(*	This FB is used for a single output solenoid 
	It uses the single input to say when Extended  	
	It starts assuming retracted and the output off.
*)
FUNCTION_BLOCK FB_Contactor_With_Single_Feedback EXTENDS FB_ComponentBase IMPLEMENTS I_Contactor
VAR
    //Output
    Output 				AT %Q* : BOOL;
//	FeedBackExtended	AT %I* : BOOL;	//This could be an sensor FB
	ExtendedSensor		:FB_DigitalSensor		:= (Name := 'Sensor', DebounceMode := E_DebounceMode.SimpleFlickerFilter, DebounceTime := T#250MS, Inverted    := FALSE, SimulationInput:= FALSE, SimulationMode := E_SensorSimulationMode.InputDriven) ;

    // Internal variables
    _ExtendRequest  : BOOL;
    _RetractRequest : BOOL;
    _Extended       : BOOL;
    _Retracted      : BOOL;
    _Extending      : BOOL;
    _Retracting     : BOOL;
    _ExtendTime     : LREAL := 1000; // Default time 1s
    _RetractTime    : LREAL := 1000; // Default time 1s

    // Timer for Extend/Retract
    Extend_TON    : TON;
    Retract_TON   : TON;
    Extend_RTRIG  : R_TRIG;
    Retract_RTRIG : R_TRIG;

    //HMI 
    Contactor_HMI : ST_Contactor_HMI;
END_VAR

METHOD PROTECTED CreateEvents
VAR_INPUT
END_VAR
SUPER^.CreateEvents();
END_METHOD

METHOD CyclicLogic
//One shot the requests
Extend_RTRIG(CLK := _ExtendRequest);
Retract_RTRIG(CLK := _RetractRequest);

//Handle Extend
IF Extend_RTRIG.Q THEN
    Output          := TRUE;
    _Extending      := TRUE;
    _Retracting     := FALSE;
    _Retracted      := FALSE;
    _RetractRequest := FALSE;
END_IF

//Handle Retract
IF Retract_RTRIG.Q THEN
    Output         := FALSE;
    _Extending     := FALSE;
    _Retracting    := TRUE;
    _Extended      := FALSE;
    _ExtendRequest := FALSE;
END_IF

//Handle the time to Extend/Retract
Extend_TON(IN := _Extending, PT := LREAL_TO_TIME(_ExtendTime));
Retract_TON(IN := _Retracting, PT := LREAL_TO_TIME(_RetractTime));
IF ExtendedSensor.Active THEN
    _Extended  := TRUE;
    _Extending := FALSE;
END_IF

IF Retract_TON.Q AND NOT ExtendedSensor.Active THEN
    _Retracted  := TRUE;
    _Retracting := FALSE;
END_IF

SUPER^.CyclicLogic();
END_METHOD

METHOD Extend
_ExtendRequest  := TRUE;
_RetractRequest := FALSE;
END_METHOD

PROPERTY Extended : BOOL
GET
Extended := _Extended;
END_GET
END_PROPERTY

PROPERTY ExtendTime : LREAL
GET
ExtendTime := _ExtendTime;
END_GET
SET
END_SET
END_PROPERTY

METHOD PROTECTED HMICommunication
VAR_INPUT
END_VAR
SUPER^.HMICommunication();

//Handle the requests to extend and retract
IF ComponentBase_HMI.Status.HMIControlAvailable THEN
    IF Contactor_HMI.Command.Extend THEN
        Extend();
    ELSIF Contactor_HMI.Command.Retract THEN
        Retract();
    END_IF
END_IF

//Update HMI status info
Contactor_HMI.Status.Extended    := _Extended;
Contactor_HMI.Status.Extending   := _Extending;
Contactor_HMI.Status.Retracted   := _Retracted;
Contactor_HMI.Status.Retracting  := _Retracting;
Contactor_HMI.Config.ExtendTime  := _ExtendTime;
Contactor_HMI.Config.RetractTime := _RetractTime;
END_METHOD

//! @summary Basic component initialization logic
METHOD PROTECTED Initialize : BOOL;

//! @description This method is called by <c>CyclicLogic()</c> as required
//Set the Contactor to retracted
IF Output THEN
    _Extended  := TRUE;
    _Retracted := FALSE;
ELSE
    _Extended  := FALSE;
    _Retracted := TRUE;
END_IF

_Extending      := FALSE;
_ExtendRequest  := FALSE;
_Retracting     := FALSE;
_RetractRequest := FALSE;

//Call base class Initialize
Initialize := SUPER^.Initialize();
END_METHOD

METHOD PROTECTED Monitoring
VAR_INPUT
END_VAR
_Busy    := _Extending OR _Retracting;
_Error   := FALSE;
_ErrorID := 0;
SUPER^.Monitoring();
END_METHOD

METHOD Retract
_ExtendRequest  := FALSE;
_RetractRequest := TRUE;
END_METHOD

PROPERTY Retracted : BOOL
GET
Retracted := _Retracted;
END_GET
END_PROPERTY

PROPERTY RetractTime : LREAL
GET
RetractTime := _RetractTime;
END_GET
SET
_RetractTime := RetractTime;
END_SET
END_PROPERTY

END_FUNCTION_BLOCK

(* stored: Version 1.1.0.1, ProductVersion 3.1.4024.15
   POU FB_Contactor_With_Single_Feedback: Id {bfc9f86d-7473-4b08-9c47-f95d13ccdae5}, SpecialFunc None
   Folder I_ComponentBase: Id {2273ad5b-ac8d-4d84-b19e-24943977fc59}
   Folder I_Contactor: Id {89231339-81c0-467b-a7c2-5ce69f410a9f}
   Folder I_CyclicFB: Id {989fbd85-70cf-447a-811a-61d4c2af51f5}
   Method CreateEvents: Id {26ac290b-88f1-466f-8ae4-f58b7a89b002}
   Method CyclicLogic: Id {8e0bcf51-f83e-4e7e-8a56-a6a8b390a3ad}
   Method Extend: Id {36a1ec48-af1d-4568-b7b9-90f73cb93cb4}
   Property Extended: Id {c2b9a74e-c7ae-4f37-8b18-09b08fc2f4fb}
   Get Get: Id {e9f55350-a9db-436f-adba-da9b7c48dbdb}
   Property ExtendTime: Id {d20af66e-b4b1-4ec2-bdc5-a99a5cb2279a}
   Get Get: Id {b3bda55b-62fc-41fc-8be8-483ad1649445}
   Set Set: Id {5bf913c0-590f-480e-8311-0d187bf1f2a7}
   Method HMICommunication: Id {48240ea5-06c3-4c68-82d4-7f47fd215c3a}
   Method Initialize: Id {4fd75c06-3e36-4e03-ace9-713e0c33b578}
   Method Monitoring: Id {9a32bee0-b1b7-435c-888b-6cc743625cd0}
   Method Retract: Id {bda24502-2f80-44e6-bfc0-f48302ba13a3}
   Property Retracted: Id {14b56551-43a5-4d92-a13d-f9712b3bd13b}
   Get Get: Id {6eb92f15-00c6-404e-a1d6-0ed0bf919be5}
   Property RetractTime: Id {6a1dece2-8998-40ed-abb9-7240a203eaca}
   Get Get: Id {b59b9704-2820-4377-a658-0afffc0b71b9}
   Set Set: Id {75cf863c-aa16-4354-be11-1e928900b6e6} *)
